PROGRAM MAIN
VAR
END_VAR

MarciaArrestoMotore();

ACTION MarciaArrestoMotore:
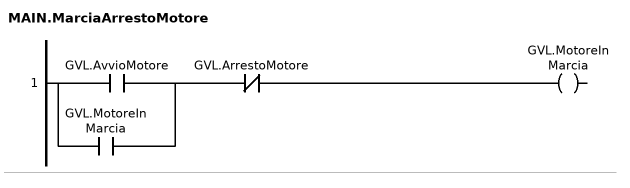
// NETWORK 1
GVL.MotoreInMarcia := (GVL.AvvioMotore OR GVL.MotoreInMarcia) AND NOT GVL.ArrestoMotore;
END_ACTION

END_PROGRAM

(* stored: Version 1.1.0.1, ProductVersion 3.1.4024.12
   POU MAIN: Id {f549e1ac-effa-45d6-85b5-ca6e4e255b2b}, SpecialFunc None
   Action MarciaArrestoMotore: Id {2921a66a-7692-437d-8326-ab5beb734472} *)
